(* PLC project SafeLOGIC-1, BrAutomation SafeDESIGNER 2.90.21.261 *)
(* stored: companyURL http://www.br-automation.com, creationDateTime Wed Sep 20 10:33:30 2017 *)

PROGRAM Main

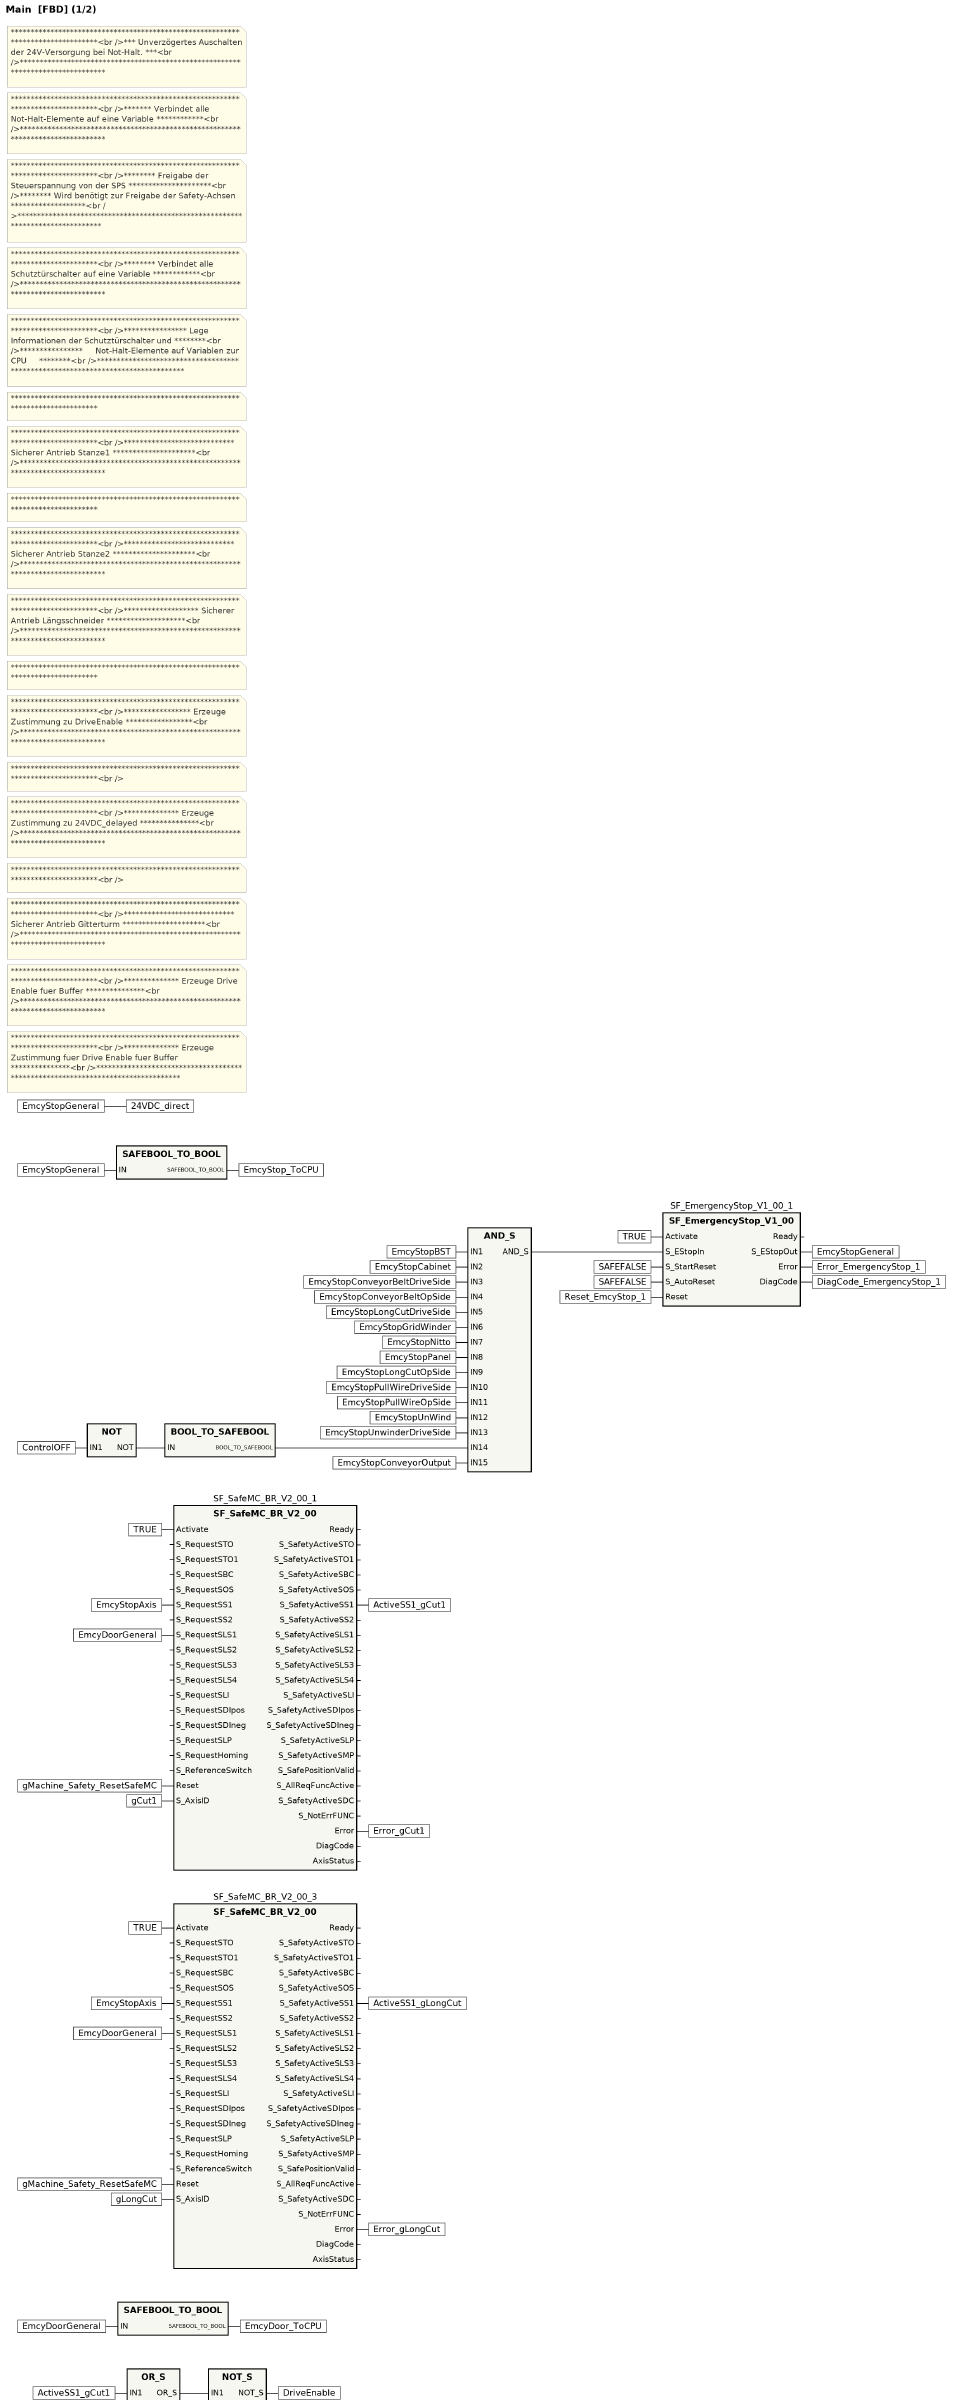
(* FBD diagram, written out as Structured Text *)
(* ********************************************************************************<br />******* Verbindet alle Not-Halt-Elemente auf eine Variable ************<br />******************************************************************************** *)
SF_EmergencyStop_V1_00_1(Activate := TRUE, S_EStopIn := AND_S(EmcyStopBST, EmcyStopCabinet, EmcyStopConveyorBeltDriveSide, EmcyStopConveyorBeltOpSide, EmcyStopLongCutDriveSide, EmcyStopGridWinder, EmcyStopNitto, EmcyStopPanel, EmcyStopLongCutOpSide, EmcyStopPullWireDriveSide, EmcyStopPullWireOpSide, EmcyStopUnWind, EmcyStopUnwinderDriveSide, BOOL_TO_SAFEBOOL(NOT ControlOFF), EmcyStopConveyorOutput), S_StartReset := SAFEFALSE, S_AutoReset := SAFEFALSE, Reset := Reset_EmcyStop_1);
Error_EmergencyStop_1 := SF_EmergencyStop_V1_00_1.Error;
DiagCode_EmergencyStop_1 := SF_EmergencyStop_V1_00_1.DiagCode;
EmcyStopGeneral := SF_EmergencyStop_V1_00_1.S_EStopOut;
EmcyStop_ToNitto := EmcyStopGeneral;
TON_S_EmcyStop_ToNitto(IN := EmcyStop_ToNitto, PT := SAFETIME#50ms);
Release_EmcyStop_ToNitto := SAFEBOOL_TO_BOOL(TON_S_EmcyStop_ToNitto.Q);
SF_EmergencyStop_V1_00_3(Activate := TRUE, S_EStopIn := AND_S(EmcyDoorBufferDriveSide, EmcyDoorBufferOpSide, EmcyUnderDoorBufferDSideLeft, EmcyUnderDoorBufferOpSideLeft, EmcyUnderDoorBufferOpSideMidd, EmcyUnderDoorBufferOpSideRight), S_StartReset := SAFEFALSE, S_AutoReset := SAFEFALSE, Reset := Reset_EmcyStop_2);
EmcyDoorBuffer := SF_EmergencyStop_V1_00_3.S_EStopOut;
Error_EmergencyStop_2 := SF_EmergencyStop_V1_00_3.Error;
DiagCode_EmergencyStop_2 := SF_EmergencyStop_V1_00_3.DiagCode;
(* ********************************************************************************<br />******** Freigabe der Steuerspannung von der SPS *********************<br />******** Wird benötigt zur Freigabe der Safety-Achsen *******************<br />******************************************************************************** *)
EmcyStopAxis := AND_S(EmcyStopGeneral, BOOL_TO_SAFEBOOL(EnabDrives_FromCPU));
(* ********************************************************************************<br />******** Verbindet alle Schutztürschalter auf eine Variable ************<br />******************************************************************************** *)
SF_EmergencyStop_V1_00_2(Activate := TRUE, S_EStopIn := AND_S(EmcyDoor1Cut1, EmcyDoor1Cut2, EmcyDoor2Cut1, EmcyDoor2Cut2, EmcyDoorBufferDriveSide, EmcyDoorBufferOpSide, EmcyDoorLongCut, EmcyDoorPBS1, EmcyUnderDoorBufferDSideLeft, EmcyUnderDoorBufferOpSideLeft, EmcyUnderDoorBufferOpSideMidd, EmcyUnderDoorBufferOpSideRight), S_StartReset := SAFEFALSE, S_AutoReset := SAFEFALSE, Reset := Reset_EmcyStop_2);
EmcyDoorGeneral := SF_EmergencyStop_V1_00_2.S_EStopOut;
Error_EmergencyStop_2 := SF_EmergencyStop_V1_00_2.Error;
DiagCode_EmergencyStop_2 := SF_EmergencyStop_V1_00_2.DiagCode;
(* ********************************************************************************<br />**************** Lege Informationen der Schutztürschalter und ********<br />****************     Not-Halt-Elemente auf Variablen zur CPU     ********<br />******************************************************************************** *)
EmcyStop_ToCPU := SAFEBOOL_TO_BOOL(EmcyStopGeneral);
(* ********************************************************************************<br />*** Unverzögertes Auschalten der 24V-Versorgung bei Not-Halt. ***<br />******************************************************************************** *)
EmcyDoor_ToCPU := SAFEBOOL_TO_BOOL(EmcyDoorGeneral);
24VDC_direct := EmcyStopGeneral;
TON_S_24VDC_direct(IN := EmcyStopGeneral, PT := SAFETIME#50ms);
Release_24VDC_direct := SAFEBOOL_TO_BOOL(TON_S_24VDC_direct.Q);
(* ******************************************************************************** *)
(* ********************************************************************************<br />**************************** Sicherer Antrieb Stanze1 *********************<br />******************************************************************************** *)
SF_SafeMC_BR_V2_00_1(Activate := TRUE, S_RequestSS1 := EmcyStopAxis, S_RequestSLS1 := EmcyDoorGeneral, Reset := gMachine_Safety_ResetSafeMC, S_AxisID := gCut1);
ActiveSS1_gCut1 := SF_SafeMC_BR_V2_00_1.S_SafetyActiveSS1;
Error_gCut1 := SF_SafeMC_BR_V2_00_1.Error;
(* ******************************************************************************** *)
(* ********************************************************************************<br />**************************** Sicherer Antrieb Stanze2 *********************<br />******************************************************************************** *)
SF_SafeMC_BR_V2_00_4(Activate := TRUE, S_RequestSS1 := EmcyStopAxis, S_RequestSLS1 := EmcyDoorGeneral, Reset := gMachine_Safety_ResetSafeMC, S_AxisID := gCut2);
ActiveSS1_gCut2 := SF_SafeMC_BR_V2_00_4.S_SafetyActiveSS1;
(* ********************************************************************************<br />**************************** Sicherer Antrieb Gitterturm *********************<br />******************************************************************************** *)
SF_SafeMC_BR_V2_00_2(Activate := TRUE, S_RequestSS1 := EmcyStopAxis, S_RequestSLS1 := EmcyDoorGeneral, Reset := gMachine_Safety_ResetSafeMC, S_AxisID := gGridFeeder);
ActiveSS1_gGridFeeder := SF_SafeMC_BR_V2_00_2.S_SafetyActiveSS1;
(* ********************************************************************************<br />******************* Sicherer Antrieb Längsschneider ********************<br />******************************************************************************** *)
SF_SafeMC_BR_V2_00_3(Activate := TRUE, S_RequestSS1 := EmcyStopAxis, S_RequestSLS1 := EmcyDoorGeneral, Reset := gMachine_Safety_ResetSafeMC, S_AxisID := gLongCut);
ActiveSS1_gLongCut := SF_SafeMC_BR_V2_00_3.S_SafetyActiveSS1;
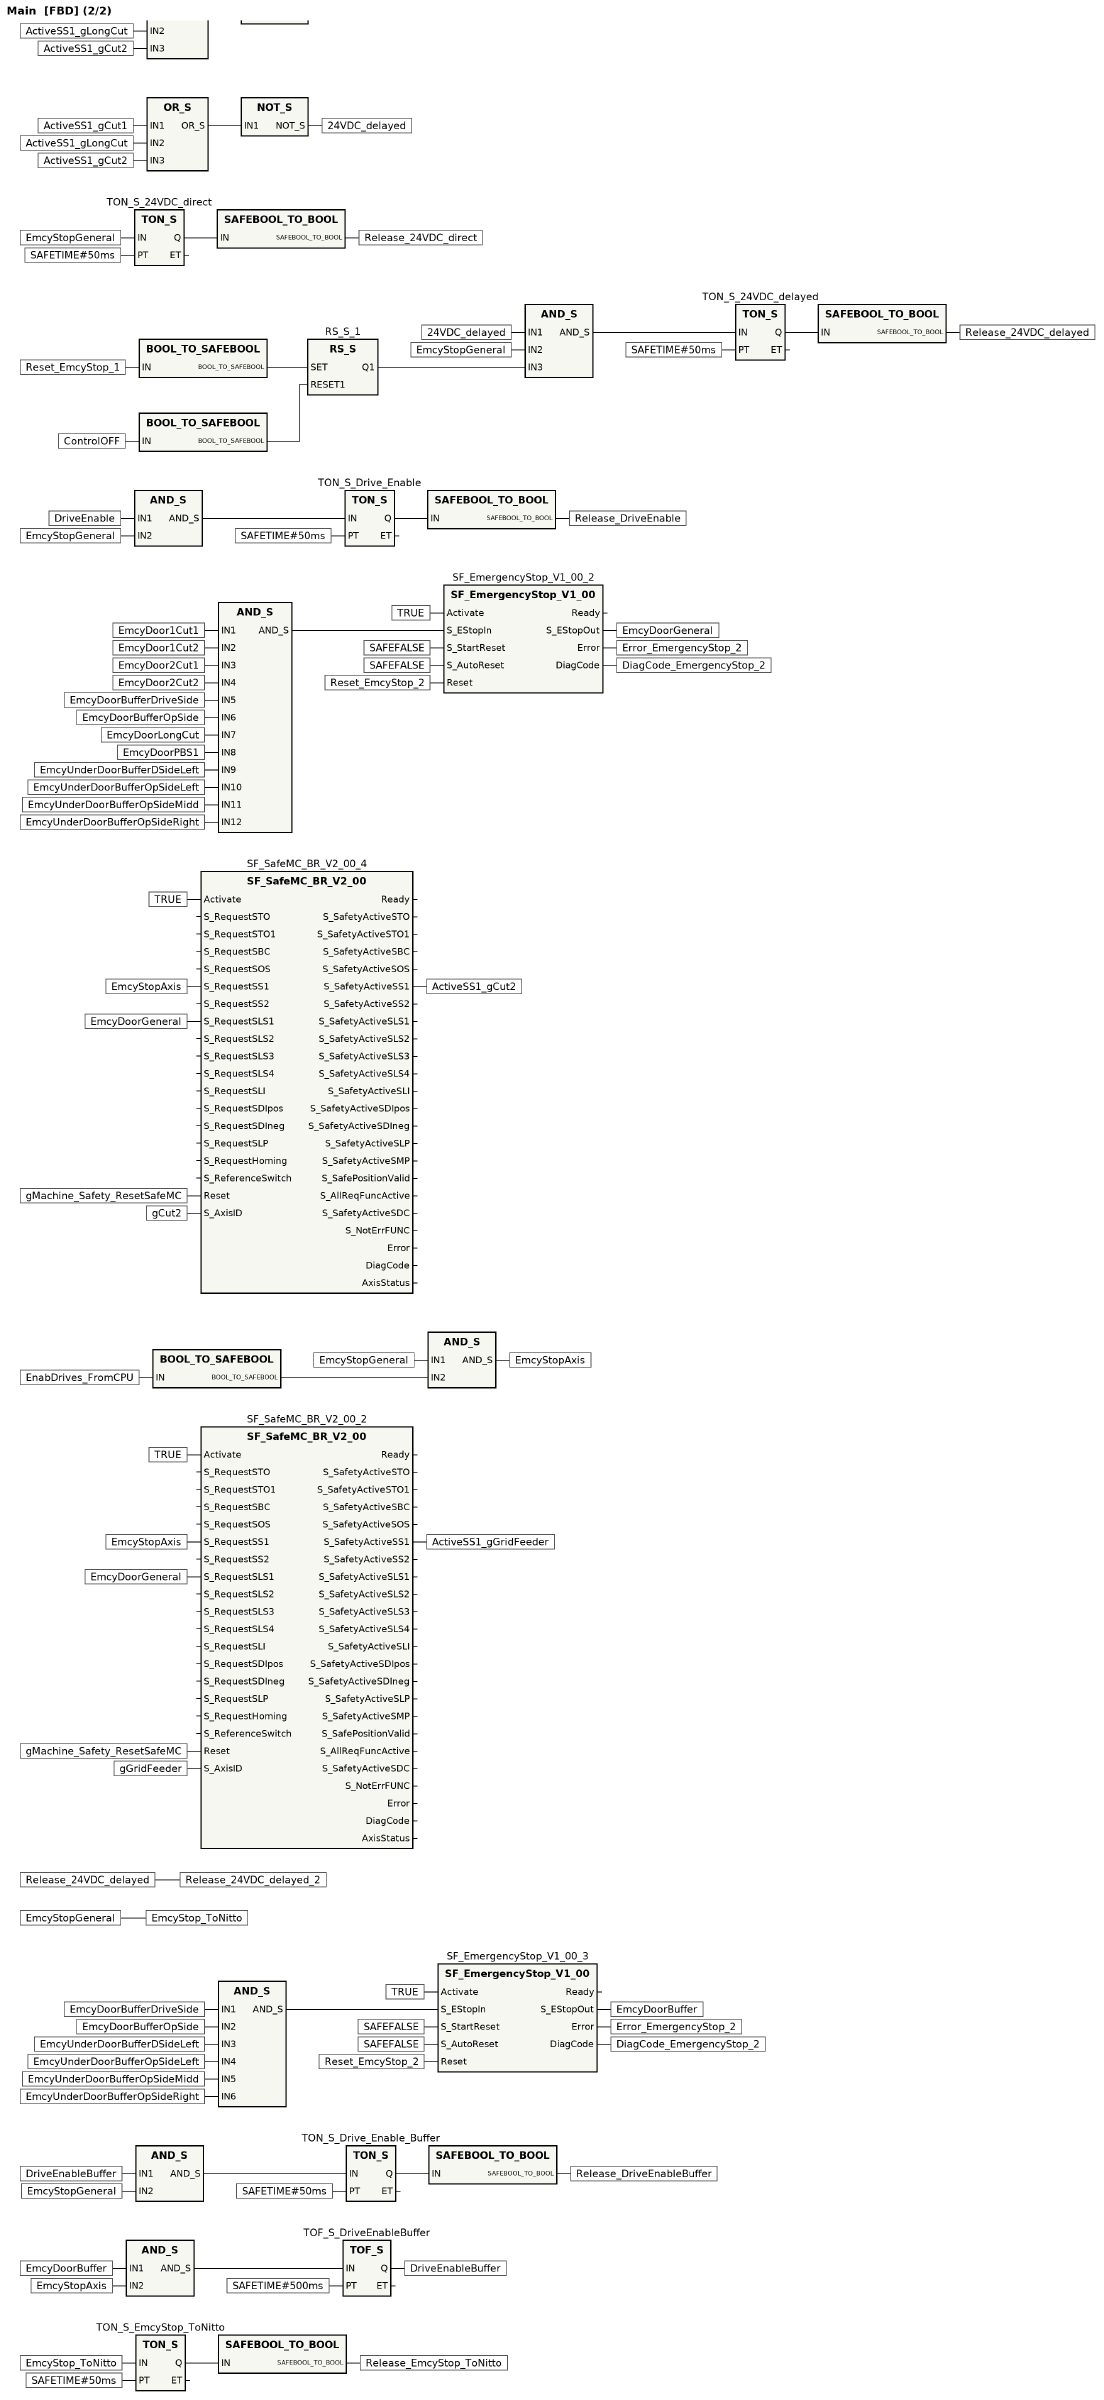
Error_gLongCut := SF_SafeMC_BR_V2_00_3.Error;
(* ******************************************************************************** *)
(* ********************************************************************************<br />***************** Erzeuge Zustimmung zu DriveEnable *****************<br />******************************************************************************** *)
DriveEnable := NOT_S(OR_S(ActiveSS1_gCut1, ActiveSS1_gLongCut, ActiveSS1_gCut2));
TON_S_Drive_Enable(IN := AND_S(DriveEnable, EmcyStopGeneral), PT := SAFETIME#50ms);
Release_DriveEnable := SAFEBOOL_TO_BOOL(TON_S_Drive_Enable.Q);
(* ********************************************************************************<br /> *)
(* ********************************************************************************<br />************** Erzeuge Zustimmung zu 24VDC_delayed ***************<br />******************************************************************************** *)
24VDC_delayed := NOT_S(OR_S(ActiveSS1_gCut1, ActiveSS1_gLongCut, ActiveSS1_gCut2));
RS_S_1(SET := BOOL_TO_SAFEBOOL(Reset_EmcyStop_1), RESET1 := BOOL_TO_SAFEBOOL(ControlOFF));
TON_S_24VDC_delayed(IN := AND_S(24VDC_delayed, EmcyStopGeneral, RS_S_1.Q1), PT := SAFETIME#50ms);
Release_24VDC_delayed := SAFEBOOL_TO_BOOL(TON_S_24VDC_delayed.Q);
Release_24VDC_delayed_2 := Release_24VDC_delayed;
(* ********************************************************************************<br /> *)
(* ********************************************************************************<br />************** Erzeuge Drive Enable fuer Buffer ***************<br />******************************************************************************** *)
TOF_S_DriveEnableBuffer(IN := AND_S(EmcyDoorBuffer, EmcyStopAxis), PT := SAFETIME#500ms);
DriveEnableBuffer := TOF_S_DriveEnableBuffer.Q;
(* ********************************************************************************<br />************** Erzeuge Zustimmung fuer Drive Enable fuer Buffer ***************<br />******************************************************************************** *)
TON_S_Drive_Enable_Buffer(IN := AND_S(DriveEnableBuffer, EmcyStopGeneral), PT := SAFETIME#50ms);
Release_DriveEnableBuffer := SAFEBOOL_TO_BOOL(TON_S_Drive_Enable_Buffer.Q);
END_PROGRAM
